SUBAPPLICATION mapping_Uebung_028 (* Analog-Eingang *)
  (* Standard: 61499-2; Description: Copyright (c) 2023 Meisterschulen am Ostbahnhof This program and the accompanying materials are made available under the terms of the Eclipse Public License 2.0 which is available at https://www.eclipse.org/legal/epl-2.0/ SPDX-License-Identifier: EPL-2.0 *)
  (* Version 1.0, 2023-10-23, Franz Höpfinger, Meisterschulen am Ostbahnhof *)
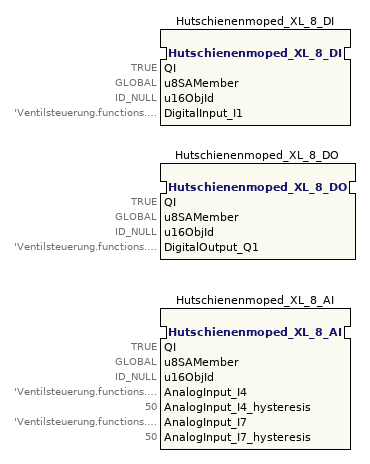
  FBS
    Hutschienenmoped_XL_8_DO : Hutschienenmoped_XL_8_DO(QI := TRUE, u8SAMember := GLOBAL, u16ObjId := ID_NULL, DigitalOutput_Q1 := 'Ventilsteuerung.functions.DigitalOutput_Q1');
    Hutschienenmoped_XL_8_DI : Hutschienenmoped_XL_8_DI(QI := TRUE, u8SAMember := GLOBAL, u16ObjId := ID_NULL, DigitalInput_I1 := 'Ventilsteuerung.functions.DigitalInput_I1');
    Hutschienenmoped_XL_8_AI : Hutschienenmoped_XL_8_AI(QI := TRUE, u8SAMember := GLOBAL, u16ObjId := ID_NULL, AnalogInput_I4 := 'Ventilsteuerung.functions.AnalogInput_I4', AnalogInput_I4_hysteresis := 50, AnalogInput_I7 := 'Ventilsteuerung.functions.AnalogInput_I7', AnalogInput_I7_hysteresis := 50);
  END_FBS
END_SUBAPPLICATION
